{attribute 'linkalways'} 
{attribute 'no_explicit_call' := 'This FB is a CLASS and must be accessed using methods or properties'}
{attribute 'enable_dynamic_creation'}
FUNCTION_BLOCK _ETcVnFilterDirection EXTENDS EnumDatatypeBase
VAR
	localData : ETcVnFilterDirection;
	activeData : REFERENCE TO ETcVnFilterDirection;
	enumBaseDatatype : _INT(localData);
END_VAR

METHOD PRIVATE AddLocalEnumeration
VAR_INPUT
	Enumeration : T_MAXSTRING;
	Value : ETcVnFilterDirection;
END_VAR
AddEnumeration(Enumeration, Value);
END_METHOD

PROPERTY PUBLIC Address : PVOID
GET
Address := ADR(activeData);
END_GET
END_PROPERTY

METHOD PUBLIC ClearReference
VAR_INPUT
END_VAR
activeData REF= localData;
SetBaseDatatypeReference();
END_METHOD

METHOD PUBLIC Clone : I_Datatype
VAR
    pClone : POINTER TO _ETcVnFilterDirection;
END_VAR
pClone := __NEW(_ETcVnFilterDirection(InitialValue := Value));
Clone := pClone^;
END_METHOD

METHOD FB_init : BOOL
VAR_INPUT
	bInitRetains : BOOL; // if TRUE, the retain variables are initialized (warm start / cold start)
	bInCopyCode : BOOL;  // if TRUE, the instance afterwards gets moved into the copy code (online change)
	InitialValue : ETcVnFilterDirection;
END_VAR
localData := InitialValue;
AddBaseDatatype(enumBaseDatatype);
ClearReference();

AddLocalEnumeration('TCVN_FD_X', ETcVnFilterDirection.TCVN_FD_X);
AddLocalEnumeration('TCVN_FD_Y', ETcVnFilterDirection.TCVN_FD_Y);
END_METHOD

PROPERTY PUBLIC Identifier : T_MAXSTRING
GET
Identifier := 'ETcVnFilterDirection';
END_GET
END_PROPERTY

METHOD IsEnumeratorValueEqual : BOOL
VAR_INPUT
	Enumerator : I_KeyValueForwardEnumerator;
END_VAR
VAR
	storedValue : ETcVnFilterDirection;
END_VAR
IF NOT Enumerator.TryGet(storedValue) THEN
	RETURN;
END_IF

IsEnumeratorValueEqual := storedValue = activeData;
END_METHOD

METHOD PUBLIC MakeReferenceTo
VAR_INPUT
	ReferenceTarget : REFERENCE TO ETcVnFilterDirection;
END_VAR
activeData REF= ReferenceTarget;
SetBaseDatatypeReference();
END_METHOD

METHOD PROTECTED SetBaseDatatypeReference
VAR_INPUT
END_VAR
enumBaseDatatype.MakeReferenceTo(activeData);
END_METHOD

PROPERTY PUBLIC Size : UDINT
GET
Size := SIZEOF(activeData);
END_GET
END_PROPERTY

METHOD TryMakeReferenceTo : BOOL
VAR_INPUT
	Target : I_Datatype;
END_VAR
VAR
	targetAsEnum : I_EnumDatatype;
	pTargetData : POINTER TO ETcVnFilterDirection;
END_VAR
IF NOT Target.TryResolveAsEnumDatatype(targetAsEnum) THEN
	RETURN;
END_IF

IF targetAsEnum.Identifier <> Identifier THEN
	RETURN;
END_IF

pTargetData := Target.Address;
activeData REF= pTargetData^;
SetBaseDatatypeReference();
TryMakeReferenceTo := TRUE;
END_METHOD

PROPERTY PUBLIC Value : ETcVnFilterDirection
GET
Value := activeData;
END_GET
SET
activeData := Value;
END_SET
END_PROPERTY

END_FUNCTION_BLOCK

(* stored: Version 1.1.0.1
   POU _ETcVnFilterDirection: Id {20e9382b-f36c-424c-bc89-3a9645896928}, SpecialFunc None
   Folder Constructor: Id {443f0271-4d17-4f4b-975d-1fb672800f68}
   Folder Private: Id {584ddeb1-00e8-469a-b824-8c9ba60b0c1b}
   Folder Protected: Id {484d0bf7-735a-4694-bbf1-d0d1b784e59e}
   Method AddLocalEnumeration: Id {9bfac190-32b7-4241-a3dc-08465a6cdf8a}
   Property Address: Id {3d85eaff-8c84-4fe1-894b-03b350cac4a8}
   Get Get: Id {a04f1091-a761-4472-9e0a-aa90aec88ec1}
   Method ClearReference: Id {d9d45623-73b6-4ddf-9c68-f2d76d232f86}
   Method Clone: Id {83485ecd-7e78-47db-8594-9bbce67b7f57}
   Method FB_init: Id {f22267bf-6c7e-41fd-a83b-4a19ca9d8c3d}
   Property Identifier: Id {dce5b4a7-f4c4-40a3-b939-72709f0d1be6}
   Get Get: Id {8357326b-5971-43c9-8c15-bf1b3706537b}
   Method IsEnumeratorValueEqual: Id {d6f2fa23-d944-4404-b6b4-977b71af7d21}
   Method MakeReferenceTo: Id {53ad012e-4717-4a4e-a103-8e0cc62334c4}
   Method SetBaseDatatypeReference: Id {b75568ee-09a5-423c-bd70-ccad5e0d4386}
   Property Size: Id {d0a61510-9e6a-4801-bf81-56389b83b13b}
   Get Get: Id {e2323f18-3ad9-4eb5-9df2-cdb9d597d715}
   Method TryMakeReferenceTo: Id {238f1ba7-4ee8-4b67-ad68-d54bbf5bbf8b}
   Property Value: Id {7a8d2af4-b7c3-473f-805f-c67818baccf7}
   Get Get: Id {65fc8dff-85a5-40ef-aec9-79e1888925dc}
   Set Set: Id {37abe5ea-b15e-40fe-a9bb-0e1ada3742e3} *)
